Staubli VAL3: GenericDetect.dtx

public bool bTaskDetOK
public num nMaxNumOfObject = 10
public num nNumOfPart = -1
num nObjectID = -1
string sDetNum
string sTASK
trsf trObjectPos
public bool bCalibrating
num nLatchedValue
